DATA_BLOCK "DB"
{ S7_Optimized_Access := 'true' }
    VAR
        inp: LREAL;
        c: LREAL;
        preset_c: TIME;
        aut_r: LREAL;
        aut_b: BOOL;
        aut_i: DINT;
        aut_tii: TupleStruct2;
        aut: BOOL;
        firstRun: BOOL;
    END_VAR
BEGIN
    firstRun := TRUE;
END_DATA_BLOCK
